# B&R Automation Studio project CrossCutterExercise
Automation Studio 4.12.4.107 SP; technology packages: Acp10Arnc0 5.24.1, mapp 5.24.1, mappView 5.24.1

## Configuration Config1

CPU 4PPC70.101G-20B, AutomationRuntime B4.93, Build 4.1.2, Safety 0.0, Vc V4.73.0

CPU 5PPC2100.BY22-000, AutomationRuntime B4.83, Build 4.1.2, Safety 0.0, Vc V4.73.0

CPU X20CP0484, AutomationRuntime B4.93, Build 4.1.2, Vc V4.72.6

### Task classes (Cpu.sw)
```
Cyclic#4:
  AxisCtrl <- SOURCE.Axis.AxisCtrl.prg
  VisuCtrl <- SOURCE.Visu.VisuCtrl.prg
  MainCtrl <- SOURCE.MainCtrl.prg
DataObjects: Acp10sys
NcDataObjects: acp10etxen <- acp10etxen.dob, gAxis01a <- gAxis01obj.gAxis01a.dob, gAxis01i <- gAxis01obj.gAxis01i.dob, gAxis02a <- gAxis02obj.gAxis02a.dob, gAxis02i <- gAxis02obj.gAxis02i.dob
Binaries: arsvcreg, udbdef, TCData, FWRules, Acp10map, acp10cfg, ashwd, ashwac, User, sysconf, asfw, arconfig, iomap, Role
Libraries: Acp10man, Acp10par, NcGlobal, Acp10_MC, sys_lib, brsystem, runtime, Acp10sim, MpAxis, MpBase, MpCom, powerlnk, astime, asbrstr, fileio, dataobj
```

### Hardware
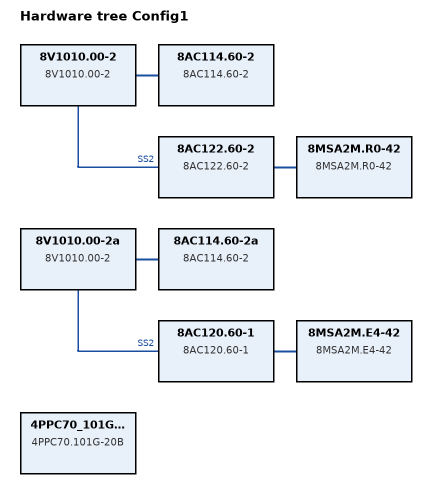
```
4PPC70_101G_20B : 4PPC70.101G-20B v1.5.4.0
  Connector IF2:
    ActivateDevice = 1
    Mode = Manual
    InternetAddress = 192.168.0.10
    SubnetMask = 255.255.255.0
    ActivateSnmp = 2
    DeviceParam = /EDDN=gei
  ConfigurationID = CrossCutterExercise_Config1
  PermanentPvSize = 2000
  RemanentGlobalPvSize = 2000
  TimerDeviceType = EPLX2X
  TimerDevice = 4PPC70_101G_20B.IF1
  TaskClassIdleTime = 2000
  FileDevice1
  FileDeviceName1 = USER
  FileDevicePath1 = USER_PATH
  KeyMappingFile = VC\4PPC70_101G_20B.dis
8AC114.60-2 : 8AC114.60-2 v1.0.0.8  [SS -> 8V1010.00-2.SS1; PLK1 -> 4PPC70_101G_20B.IF1 (NodeNumber=1) [Cable Type=PowerlinkCable, Length=10, Version=1.0.0.3]; PLK2 -> 8AC114.60-2a.PLK2 (NodeNumber=1) [Cable Type=PowerlinkCable, Length=10, Version=1.0.0.3]]
8AC114.60-2a : 8AC114.60-2 v1.0.0.8  [SS -> 8V1010.00-2a.SS1; PLK2 -> 8AC114.60-2.PLK2 (NodeNumber=2) [Cable Type=PowerlinkCable, Length=10, Version=1.0.0.3]]
8AC120.60-1 : 8AC120.60-1 v2.2.0.0  [SS -> 8V1010.00-2a.SS2]
8AC122.60-2 : 8AC122.60-2 v2.2.0.0  [SS -> 8V1010.00-2.SS2]
8MSA2M.E4-42 : 8MSA2M.E4-42 v1.0.0.0  [EC -> 8AC120.60-1.EC; MT -> 8V1010.00-2a.MT1]
8MSA2M.R0-42 : 8MSA2M.R0-42 v1.0.0.0  [EC -> 8AC122.60-2.EC; MT -> 8V1010.00-2.MT1]
8V1010.00-2 : 8V1010.00-2 v2.2.0.0
  MotionTP = Acp10Arnc0
  SinglePhaseOperation = on
  AxisIsPeriodic_r1 = on
  Period_r1 = 3600
  BothEndSwitchesAreNormallyOpen_r1 = on
  QuickStopIsNormallyOpen_r1 = on
8V1010.00-2a : 8V1010.00-2 v2.2.0.0
  MotionTP = Acp10Arnc0
  SinglePhaseOperation = on
  AxisIsPeriodic_r1 = on
  Period_r1 = 3600
  BothEndSwitchesAreNormallyOpen_r1 = on
  QuickStopIsNormallyOpen_r1 = on
```

### Acp10cfg.ncc - 4PPC70_101G_20B/Motion/Acp10cfg.ncc
```
NcConfiguration (Version=5.24.1, NcSwId=Acp10)
  ACP10CF1_typ:
    cnt_nettrc_rec_drive = 1500
    bufsize_trace_upload = 1200
    tc_nc_man_task = Cyclic #1
    glob_pv_as_ncobject = Yes
    ncsys_dl_broadcast = Yes
    ncsys_dl_acp_reset = Yes
    safemc_log_err_to_ax = Yes
    network_init:
      ncsw_init_execute = Yes
      automatic_execute = Yes
      node_nr_warning = Yes
      net_err_before_ncact = Yes
    nettrc:
      enter_parsecrec = Yes
      enter_ncaction = Yes
      save_ring_startidx = Yes
    cam_prof_download:
      cam_dat_dl_parallel = No
      tc_cam_dl_parallel = Task class for NC Manager task
    plk_if[0]:
      if_name = IF1
      tc_CycDat_PLCopen = Task class for NC Manager task
      mc_broadcast_extdat = No
```

### Acp10map.ncm - 4PPC70_101G_20B/Motion/Acp10map.ncm
```
NcMapping (NcSwId=Acp10, DisabledNodesAreHidden=False)
  NcObject gAxis02 (ModuleId=8V1010.00-2a, Type=ncAXIS, Channel=1, AcoposSimulation=Off, InitParameter=gAxis02i, AcoposParameter=gAxis02a, AdditionalData=PLCopen_ModPos="3600,1" , Disabled=FALSE, ModuleDisabled=FALSE)  // Master Axis
  NcObject gAxis01 (ModuleId=8V1010.00-2, Type=ncAXIS, Channel=1, AcoposSimulation=Off, InitParameter=gAxis01i, AcoposParameter=gAxis01a, AdditionalData=PLCopen_ModPos="3600,1" , Disabled=FALSE, ModuleDisabled=FALSE)  // Slave Axis
  NcObject 8V1010.00-2_ncV_AXIS1 (ModuleId=8V1010.00-2, Type=ncV_AXIS, Channel=1, Disabled=TRUE, ModuleDisabled=FALSE)
  NcObject 8V1010.00-2a_ncV_AXIS1 (ModuleId=8V1010.00-2a, Type=ncV_AXIS, Channel=1, Disabled=TRUE, ModuleDisabled=FALSE)
```

### Config.mpaxisbasic - 4PPC70_101G_20B/Motion/Config.mpaxisbasic
```
Element gML_Master (Type=mpaxisbasic)
```

### Config_1.mpaxisbasic - 4PPC70_101G_20B/Motion/Config_1.mpaxisbasic
```
Element gML_Slave (Type=mpaxisbasic)
  Alarms = MpAlarmX
```

### Config_4.mpaudittrail - 4PPC70_101G_20B/mappServices/Audit/Config_4.mpaudittrail
```
Element gAuditTrail (Type=mpaudittrail)
  Audit:
    Events:
      [0] = 16
      [1] = 2
      [2] = 18
    TextSource = TXT
      OutputFormat = Audit/Root
  Monitor:
    0:
      pv = ::VisuCtrl:SpeedInRPM
  Alarms = MpAlarmX
```

### Config_2.mpalarmxcore - 4PPC70_101G_20B/mappServices/Config_2.mpalarmxcore
```
Element gAlarmXCore (Type=mpalarmxcore)
  mapp.AlarmX.Core.Configuration:
    [0]:
      Name = EStopActive
      Message = Emergency Stop is Pressed
      Behavior = PersistentAlarm
```

### Config_4.mpaudittrail - 4PPC70_101G_20B/mappServices/Config_4.mpaudittrail
```
Element gAuditTrail (Type=mpaudittrail)
  Audit:
    Events:
      [0] = 16
      [1] = 2
      [2] = 18
```

### Config_5.mpcomgroup - 4PPC70_101G_20B/mappServices/Config_5.mpcomgroup
```
Element gGroup (Type=mpcomgroup)
  Linking:
    Subnodes:
      0 = gML_Master
      1 = gML_Slave
      2 = gAlarmXCore
  Alarms = MpAlarmX
Element gGroup_1 (Type=mpcomgroup)
  Linking:
    Subnodes:
      0 = gGroup
  Alarms = MpAlarmX
```

### Config_3.mpreportcore - 4PPC70_101G_20B/mappServices/Report/Config_3.mpreportcore
```
Element gReport (Type=mpreportcore)
  MpReport:
    PageLayouts:
      [0]:
        Name = Default
    Styles:
      Text:
        [0]:
          Name = Default
      Table:
        [0]:
          Name = Default
      Line:
        [0]:
          Name = Default
      Chart:
        PieChart:
          [0]:
            Name = Default
        LineChart:
          [0]:
            Name = Default
        BarChart:
          [0]:
            Name = Default
    Reports:
      [0]:
        PageLayout = Default
        [0]
```

### Config_6.mpuserx - 4PPC70_101G_20B/mappServices/User/Config_6.mpuserx
```
Element UserMgmtX (Type=mpuserx)
  ServerSettings:
    Server:
      AdditionalUserData:
        [0] = mail
        [1] = telephoneNumber
  Users:
    DefUser#1:
      id = Admin
      name = Admin
    DefUser#2:
      id = Anonymous
```

## Configuration CrossCutter

### Hardware
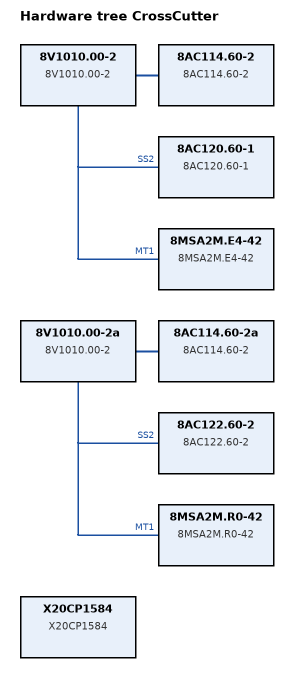
```
8AC114.60-2 : 8AC114.60-2 v1.0.0.8  [SS -> 8V1010.00-2.SS1; PLK1 -> X20CP1584.IF3 (NodeNumber=1) [Cable Type=PowerlinkCable, Length=10, Version=1.0.0.3]; PLK2 -> 8AC114.60-2a.PLK1 (NodeNumber=1) [Cable Type=PowerlinkCable, Length=10, Version=1.0.0.3]]
8AC114.60-2a : 8AC114.60-2 v1.0.0.8  [SS -> 8V1010.00-2a.SS1; PLK1 -> 8AC114.60-2.PLK2 (NodeNumber=2) [Cable Type=PowerlinkCable, Length=10, Version=1.0.0.3]]
8AC120.60-1 : 8AC120.60-1 v2.2.0.0  [SS -> 8V1010.00-2.SS2]
8AC122.60-2 : 8AC122.60-2 v2.2.0.0  [SS -> 8V1010.00-2a.SS2]
8MSA2M.E4-42 : 8MSA2M.E4-42 v1.0.0.0  [MT -> 8V1010.00-2.MT1]
8MSA2M.R0-42 : 8MSA2M.R0-42 v1.0.0.0  [MT -> 8V1010.00-2a.MT1]
8V1010.00-2 : 8V1010.00-2 v2.2.0.0
  MotionTP = Acp10Arnc0
  SinglePhaseOperation = on
  AxisIsPeriodic_r1 = on
  Period_r1 = 3600
  BothEndSwitchesAreNormallyOpen_r1 = on
  QuickStopIsNormallyOpen_r1 = on
8V1010.00-2a : 8V1010.00-2 v2.2.0.0
  MotionTP = Acp10Arnc0
  SinglePhaseOperation = on
  AxisIsPeriodic_r1 = on
  Period_r1 = 3600
  BothEndSwitchesAreNormallyOpen_r1 = on
  QuickStopIsNormallyOpen_r1 = on
X20CP1584 : X20CP1584 v1.10.0.0
  Connector IF2:
    ActivateDevice = 1
    Mode = Manual
    InternetAddress = 192.168.0.12
    SubnetMask = 255.255.255.0
    ActivateSnmp = 2
  ConfigurationID = CamAutomat_CrossCutter
  Simulation = 1
  TimerDeviceType = EPLX2X
  TimerDevice = X20CP1584.IF3
  TaskClassIdleTime = 2000
  FileDevice1
  FileDeviceName1 = USER
  FileDevicePath1 = USER_PATH
```

## Logical view

Binary libraries used (declarations not repeated): operator, runtime, astime, AsIecCon, sys_lib, brsystem, Acp10man, Acp10par, NcGlobal, Acp10sim 5.24.1, Acp10_MC, MpAxis 1.87.0, MpBase, MpCom 5.24.1, MpAlarmX, MpData, FileIO, DataObj, MpAudit 5.24.1, MpServer 5.24.0, MpUserX 5.24.1, MpReport 5.24.1

### Global.var - Global variables
```iecst
VAR
	gAxis01 : ACP10AXIS_typ; (*Slave Axis*)
	gAxis02 : ACP10AXIS_typ; (*Master Axis*)
	gVAxis01 : ACP10VAXIS_typ; (*Virtual Axis*)
	gVAxis02 : ACP10VAXIS_typ; (*Virtual Axis*)
	MpAxisSlave : MpAxisBasic; (*FB for Slave*)
	MpAxisMaster : MpAxisBasic; (*FB for Master*)
	MpAxisCamSequencer_0 : MpAxisCamSequencer; (*Cam Sequencer FB*)
	CamSeqPara : MpAxisCamSequencerParType; (*Cam Sequence Parameter*)
	SlavePara : MpAxisBasicParType; (*Slave Axis Parameter*)
	MasterPara : MpAxisBasicParType; (*Master Axis Parameter*)
END_VAR
```


### Data object Logical/acp10etxen (Ett)

- acp10etxen.ett (not shown)

### Package Logical/gAxis01obj - gAxis03obj

### gAxis01i.ax
```
InitParameter (Version=5.24.1, NcSwId=Acp10)
  ACP10AXIS_typ:
    dig_in:
      level:
        reference = ncACTIV_HI + ncFORCE
        pos_hw_end = ncACTIV_HI + ncFORCE
        neg_hw_end = ncACTIV_HI + ncFORCE
        trigger1 = ncACTIV_HI
        trigger2 = ncACTIV_HI
    encoder_if:
      parameter:
        count_dir = ncINVERSE
        scaling:
          load:
            units = 3600
            rev_motor = 1
    limit:
      parameter:
        v_pos = 50000.0
        v_neg = 50000.0
        a1_pos = 120000.0
        a2_pos = 120000.0
        a1_neg = 120000.0
        a2_neg = 120000.0
        t_jolt = 0.02
        t_in_pos = 0
        pos_sw_end = 2000000000
        neg_sw_end = -2000000000
        ds_warning = 500
        ds_stop = 1000
        a_stop = 1.0e30
        dv_stop = 0
        dv_stop_mode = ncOFF
    controller:
      mode = ncPOSITION
      position:
        kv = 50
        tn = 0
        t_predict = 0.0004
        t_total = 0.0004
        p_max = 1.0e30
        i_max = 0
      speed:
        kv = 0.2
        tn = 0
        t_filter = 0.0
        isq_filter1:
          type = ncOFF
          a0 = 0.0
          a1 = 0.0
          b0 = 0.0
          b1 = 0.0
          b2 = 0.0
          c0_par_id = 0
          c1_par_id = 0
        isq_filter2:
          type = ncOFF
          a0 = 0.0
          a1 = 0.0
          b0 = 0.0
          b1 = 0.0
          b2 = 0.0
          c0_par_id = 0
          c1_par_id = 0
        isq_filter3:
          type = ncOFF
          a0 = 0.0
          a1 = 0.0
          b0 = 0.0
          b1 = 0.0
          b2 = 0.0
          c0_par_id = 0
          c1_par_id = 0
      uf:
        type = ncLINEAR + ncCORRECTION
        auto_config = ncMOTOR_PAR
        u0 = 0
        un = 0
        fn = 50.0
        k_f_slip = 0
      ff:
        mode = ncSTANDARD
        torque_load = 0.0
        torque_pos = 0.0
        torque_neg = 0.0
        kv_torque = 0.0
        inertia = 0.0
        t_filter_a = 0.0
      fb:
        mode = ncSTANDARD
        speed_mix_ratio = 0.0
        speed_kv = 0.2
      model:
        mass1:
          inertia = 0
          viscous_friction = 0
        mass2:
          inertia = 0
          viscous_friction = 0
          stiffness = 0
          damping = 0
    move:
      stop:
        parameter[0]:
          decel_ramp = ncA_LIMIT
          controller = ncON
        parameter[1]:
          decel_ramp = ncA_LIMIT
          controller = ncON
        parameter[2]:
          decel_ramp = ncA_LIMIT
          controller = ncON
        parameter[3]:
          decel_ramp = ncA_LIMIT
          controller = ncON
        quickstop:
          decel_ramp = ncA_LIMIT
          t_jolt = 0
        drive_error:
          decel_ramp = ncA_LIMIT
      homing:
        parameter:
          s = 0
          v_switch = 5000
          v_trigger = 500
          a = 50000
          mode = ncDIRECT
          edge_sw = ncPOSITIVE
          start_dir = ncPOSITIVE
          trigg_dir = ncPOSITIVE
          ref_pulse = ncOFF
          fix_dir = ncOFF
          tr_s_block = 0
          torque_lim = 0
          ds_block = 0
          ds_stop = 0
      basis:
        parameter:
          v_pos = 5000
          v_neg = 5000
          a1_pos = 50000
          a2_pos = 50000
          a1_neg = 50000
          a2_neg = 50000
    message:
      text:
        parameter:
          format = ncBREAK
          columns = 80
          data_modul = acp10etxen
```

### Package Logical/gAxis02obj - gAxis04obj

### gAxis02i.ax
```
InitParameter (Version=5.24.1, NcSwId=Acp10)
  ACP10AXIS_typ:
    dig_in:
      level:
        reference = ncACTIV_HI + ncFORCE
        pos_hw_end = ncACTIV_HI + ncFORCE
        neg_hw_end = ncACTIV_HI + ncFORCE
        trigger1 = ncACTIV_HI
        trigger2 = ncACTIV_HI
    encoder_if:
      parameter:
        count_dir = ncINVERSE
        scaling:
          load:
            units = 3600
            rev_motor = 1
    limit:
      parameter:
        v_pos = 50000.0
        v_neg = 50000.0
        a1_pos = 120000.0
        a2_pos = 120000.0
        a1_neg = 120000.0
        a2_neg = 120000.0
        t_jolt = 0.02
        t_in_pos = 0
        pos_sw_end = 2000000000
        neg_sw_end = -2000000000
        ds_warning = 500
        ds_stop = 1000
        a_stop = 1.0e30
        dv_stop = 0
        dv_stop_mode = ncOFF
    controller:
      mode = ncPOSITION
      position:
        kv = 50
        tn = 0
        t_predict = 0.0044
        t_total = 0.0044
        p_max = 1.0e30
        i_max = 0
      speed:
        kv = 0.2
        tn = 0
        t_filter = 0.0
        isq_filter1:
          type = ncOFF
          a0 = 0.0
          a1 = 0.0
          b0 = 0.0
          b1 = 0.0
          b2 = 0.0
          c0_par_id = 0
          c1_par_id = 0
        isq_filter2:
          type = ncOFF
          a0 = 0.0
          a1 = 0.0
          b0 = 0.0
          b1 = 0.0
          b2 = 0.0
          c0_par_id = 0
          c1_par_id = 0
        isq_filter3:
          type = ncOFF
          a0 = 0.0
          a1 = 0.0
          b0 = 0.0
          b1 = 0.0
          b2 = 0.0
          c0_par_id = 0
          c1_par_id = 0
      uf:
        type = ncLINEAR + ncCORRECTION
        auto_config = ncMOTOR_PAR
        u0 = 0
        un = 0
        fn = 50.0
        k_f_slip = 0
      ff:
        mode = ncSTANDARD
        torque_load = 0.0
        torque_pos = 0.0
        torque_neg = 0.0
        kv_torque = 0.0
        inertia = 0.0
        t_filter_a = 0.0
      fb:
        mode = ncSTANDARD
        speed_mix_ratio = 0.0
        speed_kv = 2.0
      model:
        mass1:
          inertia = 0
          viscous_friction = 0
        mass2:
          inertia = 0
          viscous_friction = 0
          stiffness = 0
          damping = 0
    move:
      stop:
        parameter[0]:
          decel_ramp = ncA_LIMIT
          controller = ncON
        parameter[1]:
          decel_ramp = ncA_LIMIT
          controller = ncON
        parameter[2]:
          decel_ramp = ncA_LIMIT
          controller = ncON
        parameter[3]:
          decel_ramp = ncA_LIMIT
          controller = ncON
        quickstop:
          decel_ramp = ncA_LIMIT
          t_jolt = 0
        drive_error:
          decel_ramp = ncA_LIMIT
      homing:
        parameter:
          s = 0
          v_switch = 5000
          v_trigger = 500
          a = 50000
          mode = ncDIRECT
          edge_sw = ncPOSITIVE
          start_dir = ncPOSITIVE
          trigg_dir = ncPOSITIVE
          ref_pulse = ncOFF
          fix_dir = ncOFF
          tr_s_block = 0
          torque_lim = 0
          ds_block = 0
          ds_stop = 0
      basis:
        parameter:
          v_pos = 5000
          v_neg = 5000
          a1_pos = 50000
          a2_pos = 50000
          a1_neg = 50000
          a2_neg = 50000
    message:
      text:
        parameter:
          format = ncBREAK
          columns = 80
          data_modul = acp10etxen
```

### Main.typ
```iecst
TYPE
	Main_typ : 	STRUCT
		Cmd : MainCmd_typ;
		Status : MainStatus_typ;
	END_STRUCT;
	MainCmd_typ : 	STRUCT
		bStart : BOOL;
		bStop : BOOL;
		bEStop : BOOL;
	END_STRUCT;
	MainStatus_typ : 	STRUCT
	END_STRUCT;
END_TYPE
```

### Program Logical/SOURCE/MainCtrl (IEC)

#### Types.typ
```iecst
TYPE
	eMainState :
		(
		WAIT,
		SELECT_MODE,
		SINGLE_BLADE,
		DUAL_BLADE,
		ERROR
		);
END_TYPE
```

#### Variables.var
```iecst
VAR
	MainState : eMainState;
END_VAR
```

#### Main.st
```iecst
(*|ŻŻŻŻŻŻŻŻŻŻŻŻŻŻŻŻŻŻŻŻŻŻŻŻŻŻŻŻŻŻŻŻŻŻŻŻŻŻŻŻŻŻŻŻŻŻŻŻŻŻŻŻŻŻŻŻŻŻŻŻŻŻŻŻŻŻŻŻŻŻŻŻŻŻŻŻŻŻŻŻŻŻŻŻŻŻŻŻŻŻŻŻŻŻŻŻŻŻŻŻŻŻŻŻŻŻŻŻŻŻ|*)
(*| Copyright      :-  B&R Industrial Automation GmbH                                                            |*)
(*| Contact Person :-   salis                                                                          		     |*)
(*|——————————————————————————————————————————————————————————————————————————————————————————————————————————————|*)
(*| System       :-  Cross Cutter                                                                                |*)
(*| Task Name    :-  MainCtrl.st                                                                                 |*)
(*| Auther Name  :-   salis                                                                                      |*)
(*| Created Date :-  April 28, 2024/10:21 AM                                                                     |*)
(*| AS Version   :-  AS 4.12.4.107 SP                                                                            |*)
(*|——————————————————————————————————————————————————————————————————————————————————————————————————————————————|*)
(*| Description  :-  Main Control and Mode Selection Logic                                                       |*)
(*|                                                                                                              |*)
(*|——————————————————————————————————————————————————————————————————————————————————————————————————————————————|*)
(*| Version :-         V 1.0                      salis                                                          |*)
(*|——————————————————————————————————————————————————————————————————————————————————————————————————————————————|*)
PROGRAM _INIT

END_PROGRAM

PROGRAM _CYCLIC
	(********************************* State Machine for Main Control and Mode Selection ***************************************)

	CASE MainState OF
		WAIT:

			IF Main.Cmd.bStart THEN
				MainState := SELECT_MODE;
			END_IF

		SELECT_MODE:
			IF Main.Cmd.bSingleBlade THEN
				MainState := SINGLE_BLADE;
			ELSIF Main.Cmd.bDoubleBlade THEN
				MainState := DUAL_BLADE;
			END_IF
			MpAxisMaster.Update := FALSE;
			MpAxisSlave.Update := FALSE;

		SINGLE_BLADE:
			Main.Cmd.bDoubleBlade := FALSE;
			Axis.Cmd.bDoubleBlade := FALSE;
			Main.Cmd.bSingleBlade := FALSE;
			Axis.Cmd.bSingleBlade := TRUE;
			MpAxisMaster.Update := TRUE;
			MpAxisSlave.Update := TRUE;
			IF MpAxisMaster.UpdateDone AND MpAxisSlave.UpdateDone THEN
				MainState := SELECT_MODE;
			END_IF

		DUAL_BLADE:
			Main.Cmd.bSingleBlade := FALSE;
			Axis.Cmd.bSingleBlade := FALSE;
			Main.Cmd.bDoubleBlade := FALSE;
			Axis.Cmd.bDoubleBlade := TRUE;
			MpAxisMaster.Update := TRUE;
			MpAxisSlave.Update := TRUE;
			IF MpAxisMaster.UpdateDone AND MpAxisSlave.UpdateDone THEN
				MainState := SELECT_MODE;
			END_IF
	END_CASE;

END_PROGRAM

PROGRAM _EXIT

END_PROGRAM
```

### Axis.typ
```iecst
TYPE
	Axis_typ : 	STRUCT
		Cmd : AxisCmd_typ;
		Para : AxisPara_typ;
	END_STRUCT;
	AxisCmd_typ : 	STRUCT
		bStart : BOOL;
		bHome : BOOL;
		bStop : BOOL;
		bEStop : BOOL;
	END_STRUCT;
	AxisPara_typ : 	STRUCT
		gMachineSpeed : USINT;
	END_STRUCT;
END_TYPE
```

### Program Logical/SOURCE/Axis/AxisCtrl (IEC)

#### Main.st - Init, cyclic, exit code
```iecst
PROGRAM _INIT
	(* Insert code here *)
	MasterPara.Acceleration := 5000;
	MasterPara.Deceleration := 10000;

	MasterPara.Position := 0;

	SlavePara.Acceleration := 5000;
	SlavePara.Deceleration := 10000;

	SlavePara.Position := 0;;

END_PROGRAM

PROGRAM _CYCLIC
	(* Insert code here *)

	MpAxisMaster.MpLink := ADR(gML_Master);
	MpAxisMaster.Enable := TRUE;
	MpAxisMaster.Parameters := ADR(MasterPara);
	MpAxisMaster.Axis := ADR(gAxis02);
	MpAxisMaster();

	MpAxisSlave.MpLink := ADR(gML_Slave);
	MpAxisSlave.Enable := TRUE;
	MpAxisSlave.Parameters := ADR(SlavePara);
	MpAxisSlave.Axis := ADR(gAxis01);
	MpAxisSlave();

	SingleBladeCam;

	MpAxisCamSequencer_0.MpLink := ADR(gML_Slave);
	MpAxisCamSequencer_0.MpLinkMaster := ADR(gML_Master);
	MpAxisCamSequencer_0.Enable := TRUE;
	MpAxisCamSequencer_0.Parameters := ADR(CamSeqPara);
	MpAxisCamSequencer_0();

	IF Axis.Cmd.bHome THEN
		MasterPara.Direction := mpAXIS_DIR_SHORTEST_WAY;
		SlavePara.Direction := mpAXIS_DIR_SHORTEST_WAY;
		MasterPara.Velocity := 1200;
		SlavePara.Velocity := 1200;
	ELSE
		MasterPara.Direction := mpAXIS_DIR_POSITIVE;
		SlavePara.Direction := mpAXIS_DIR_POSITIVE;
		MasterPara.Velocity := 3600;
		SlavePara.Velocity := 3600;
	END_IF

//	IF (MpAxisMaster.Position <= 1560) AND (MpAxisMaster.Position >= 2060) THEN
//		MpAxisMaster.Power := FALSE;
//		MpAxisSlave.Power := FALSE;
//	ELSIF MpAxisMaster.Active AND MpAxisSlave.Active THEN
//		MpAxisMaster.Power := TRUE;
//		MpAxisSlave.Power := TRUE;
//	END_IF

	CASE AxisHomeState OF
		WAIT:
			IF (MpAxisMaster.Power = TRUE) AND (MpAxisSlave.Power = TRUE) THEN
				IF Axis.Cmd.bHome THEN
					AxisHomeState := HOME;
				END_IF
			END_IF
		HOME:
			MpAxisCamSequencer_0.StartSequence := FALSE;
			MpAxisMaster.MoveAbsolute := TRUE;
			MpAxisSlave.MoveAbsolute := TRUE;
			IF (MpAxisMaster.Position = MasterPara.Position) AND (MpAxisSlave.Position = SlavePara.Position) THEN
				AxisHomeState := HOMING_ACTIVE;
			END_IF

		HOMING_ACTIVE:
			MpAxisMaster.MoveAbsolute := FALSE;
			MpAxisSlave.MoveAbsolute := FALSE;
			MpAxisMaster.Home := TRUE;
			MpAxisSlave.Home := TRUE;
			IF MpAxisMaster.IsHomed AND MpAxisSlave.IsHomed THEN
				AxisHomeState := HOME_OK;
			END_IF

		HOME_OK:
			MpAxisCamSequencer_0.StartSequence := TRUE;
			Axis.Cmd.bHome := FALSE;
			MpAxisMaster.MoveAbsolute := FALSE;
			MpAxisSlave.MoveAbsolute := FALSE;
			MpAxisMaster.Home := FALSE;
			MpAxisSlave.Home := FALSE;
			AxisHomeState := WAIT;

	END_CASE;

END_PROGRAM

PROGRAM _EXIT
	(* Insert code here *)

END_PROGRAM
```

#### Types.typ - Local data types
```iecst
TYPE
	eAxisHome :
		(
		WAIT,
		HOMING_ACTIVE,
		HOME,
		HOME_OK,
		ERROR
		);
END_TYPE
```

#### Variables.var - Local variables
```iecst
VAR
	AxisHomeState : eAxisHome;
	Axis : Axis_typ;
END_VAR
```

#### SingleBladeCam.st - Cam logic for single blade cross cutter
```iecst
ACTION SingleBladeCam:
	CamSeqPara.Configuration.Master 			:= ADR(gAxis02);
	CamSeqPara.Configuration.MasterParID 		:= ACP10PAR_PCTRL_S_ACT;

	(** Event 0 - WAIT FOR TRIGGER **)
	CamSeqPara.Configuration.State[0].Event[0].Type 				:= ncST_END; //Trigger
	CamSeqPara.Configuration.State[0].Event[0].Attribute		 	:= ncST_END; //Reaction
	CamSeqPara.Configuration.State[0].Event[0].NextState 			:= 1; //Next State
	(*************************** STATE 1 ****************************)
	CamSeqPara.Configuration.State[1].CamProfileIndex 		  		:= 16#FFFE;
	CamSeqPara.Configuration.State[1].MasterFactor 					:= 1; //Master Dist.
	CamSeqPara.Configuration.State[1].SlaveFactor 					:= 1; //Slave Dist.

	CamSeqPara.Configuration.State[1].CompMode   	 				:= ncONLYCOMP;
	CamSeqPara.Configuration.State[1].MasterCompDistance			:= 1620; //Master Dist.
	CamSeqPara.Configuration.State[1].SlaveCompDistance				:= 1620; //Slave Dist.

	(** Event **)
	CamSeqPara.Configuration.State[1].Event[0].Type 				:= ncST_END; //Trigger
	CamSeqPara.Configuration.State[1].Event[0].Attribute 			:= ncST_END; //Reaction
	CamSeqPara.Configuration.State[1].Event[0].NextState 			:= 2; //Next State

	(*************************** STATE 2 ****************************)
	CamSeqPara.Configuration.State[2].CamProfileIndex 				:= 16#FFFF;
	CamSeqPara.Configuration.State[2].MasterFactor 					:= 360;  //Master Dist.
	CamSeqPara.Configuration.State[2].SlaveFactor 					:= -360; //Slave Dist.

	(** Event **)
	CamSeqPara.Configuration.State[2].Event[0].Type 				:= ncST_END; //Trigger
	CamSeqPara.Configuration.State[2].Event[0].Attribute 			:= ncST_END; //Reaction
	CamSeqPara.Configuration.State[2].Event[0].NextState 			:= 3; //Next State

	(*************************** STATE 3 ****************************)
	CamSeqPara.Configuration.State[3].CamProfileIndex 				:= 16#FFFE;
	CamSeqPara.Configuration.State[3].MasterFactor 					:= 1; //Master Dist.
	CamSeqPara.Configuration.State[3].SlaveFactor 					:= 1; //Slave Dist.

	CamSeqPara.Configuration.State[3].CompMode   	 				:= ncONLYCOMP;
	CamSeqPara.Configuration.State[3].MasterCompDistance			:= 1620; //Master Dist.
	CamSeqPara.Configuration.State[3].SlaveCompDistance				:= 1620; //Slave Dist.

	(** Event **)
	CamSeqPara.Configuration.State[3].Event[0].Type 				:= ncST_END; //Trigger
	CamSeqPara.Configuration.State[3].Event[0].Attribute 			:= ncST_END; //Reaction
	CamSeqPara.Configuration.State[3].Event[0].NextState 			:= 1; //Next State
END_ACTION
```

#### DoubleBladeCam.st - Cam logic for Double blade cross cutter
```iecst
ACTION DoubleBladeCam:

	CamSeqPara.Configuration.Master 			:= ADR(gAxis02);
	CamSeqPara.Configuration.MasterParID 		:= ACP10PAR_PCTRL_S_ACT;

	(** Event 0 - WAIT FOR TRIGGER **)
	CamSeqPara.Configuration.State[0].Event[0].Type 				:= ncST_END; //Trigger
	CamSeqPara.Configuration.State[0].Event[0].Attribute		 	:= ncST_END; //Reaction
	CamSeqPara.Configuration.State[0].Event[0].NextState 			:= 1; //Next State
	(*************************** STATE 1 ****************************)
	CamSeqPara.Configuration.State[1].CamProfileIndex 		  		:= 16#FFFE;
	CamSeqPara.Configuration.State[1].MasterFactor 					:= 1; //Master Dist.
	CamSeqPara.Configuration.State[1].SlaveFactor 					:= 1; //Slave Dist.

	CamSeqPara.Configuration.State[1].CompMode   	 				:= ncONLYCOMP;
	CamSeqPara.Configuration.State[1].MasterCompDistance			:= 1580; //Master Dist.
	CamSeqPara.Configuration.State[1].SlaveCompDistance				:= 1580; //Slave Dist.

	(** Event **)
	CamSeqPara.Configuration.State[1].Event[0].Type 				:= ncST_END; //Trigger
	CamSeqPara.Configuration.State[1].Event[0].Attribute 			:= ncST_END; //Reaction
	CamSeqPara.Configuration.State[1].Event[0].NextState 			:= 2; //Next State

	(*************************** STATE 2 ****************************)
	CamSeqPara.Configuration.State[2].CamProfileIndex 				:= 16#FFFF;
	CamSeqPara.Configuration.State[2].MasterFactor 					:= 400;  //Master Dist.
	CamSeqPara.Configuration.State[2].SlaveFactor 					:= -400; //Slave Dist.

	(** Event **)
	CamSeqPara.Configuration.State[2].Event[0].Type 				:= ncST_END; //Trigger
	CamSeqPara.Configuration.State[2].Event[0].Attribute 			:= ncST_END; //Reaction
	CamSeqPara.Configuration.State[2].Event[0].NextState 			:= 0; //Next State

	(*************************** STATE 3 ****************************)
	CamSeqPara.Configuration.State[3].CamProfileIndex 				:= 16#FFFE;
	CamSeqPara.Configuration.State[3].MasterFactor 					:= 1; //Master Dist.
	CamSeqPara.Configuration.State[3].SlaveFactor 					:= 1; //Slave Dist.

	CamSeqPara.Configuration.State[3].CompMode   	 				:= ncONLYCOMP;
	CamSeqPara.Configuration.State[3].MasterCompDistance			:= 1620; //Master Dist.
	CamSeqPara.Configuration.State[3].SlaveCompDistance				:= 1620; //Slave Dist.

	(** Event **)
	CamSeqPara.Configuration.State[3].Event[0].Type 				:= ncST_END; //Trigger
	CamSeqPara.Configuration.State[3].Event[0].Attribute 			:= ncST_END; //Reaction
	CamSeqPara.Configuration.State[3].Event[0].NextState 			:= 4; //Next State

	(*************************** STATE 4 ****************************)
	CamSeqPara.Configuration.State[4].CamProfileIndex 				:= 16#FFFF;
	CamSeqPara.Configuration.State[4].MasterFactor 					:= 360;  //Master Dist.
	CamSeqPara.Configuration.State[4].SlaveFactor 					:= -360; //Slave Dist.

	(** Event **)
	CamSeqPara.Configuration.State[4].Event[0].Type 				:= ncST_END; //Trigger
	CamSeqPara.Configuration.State[4].Event[0].Attribute 			:= ncST_END; //Reaction
	CamSeqPara.Configuration.State[4].Event[0].NextState 			:= 1; //Next State
END_ACTION
```

### Axis.var - not listed in the package file held
```iecst
VAR
	Axis : Axis_typ;
END_VAR
VAR CONSTANT
	SPositionSingle : INT := 3550;
	MPositionSingle : INT := 3450;
	SlaveOffsetSingle : INT := 0;
	MasterOffsetSingle : INT := 0;
	MUpPositionDouble : INT := 825;
	SPositionDouble : INT := 2225;
	MDownPositionDouble : INT := 2625;
	MasterUpOffsetDouble : INT := 825;
	MasterDownOffsetDouble : INT := 2625;
	HomingVelocity : INT := 1200;
	MUpPosLimit1 : INT := 1480;
	MUpPosLimit2 : INT := 3501;
	MUpNegLimit1 : INT := 0;
	MUpNegLimit2 : INT := 3599;
	MDownNegLimit : INT := 1940;
	MDownPosLimit : INT := 3500;
	MCutRegionNegLimit1 : INT := 1480;
	MCutRegionPosLimit1 : INT := 1940;
	MCutRegionNegLimit2 : INT := 3280;
	MCutRegionPosLimit2 : INT := 3599;
	MCutRegionPosLimit3 : INT := 1;
	MCutRegionNegLimit3 : INT := 150;
	RunDeceleration : UDINT := 72000;
	RunAcceleration : UDINT := 72000;
	HomeAcceleration : UDINT := 3600;
	HomeVelocity : UDINT := 720;
	JogVelocity : UDINT := 7200;
END_VAR
```

- Visualisation Logical/SOURCE/Visu (not shown)

### Main.var - not listed in the package file held
```iecst
VAR
	Main : Main_typ;
	MachineStatus : STRING[80];
END_VAR
```

### Program Logical/SOURCE/Alarm/AlarmCtrl (IEC) - Program for Alarm

#### Variables.var
```iecst
VAR
	MpAlarm : MpAlarmXCore;
END_VAR
```

#### Main.st
```iecst
(*|ŻŻŻŻŻŻŻŻŻŻŻŻŻŻŻŻŻŻŻŻŻŻŻŻŻŻŻŻŻŻŻŻŻŻŻŻŻŻŻŻŻŻŻŻŻŻŻŻŻŻŻŻŻŻŻŻŻŻŻŻŻŻŻŻŻŻŻŻŻŻŻŻŻŻŻŻŻŻŻŻŻŻŻŻŻŻŻŻŻŻŻŻŻŻŻŻŻŻŻŻŻŻŻŻŻŻŻŻŻŻ|*)
(*| Copyright      :-  B&R Industrial Automation GmbH                                                            |*)
(*| Contact Person :-   salis                                                                          		     |*)
(*|——————————————————————————————————————————————————————————————————————————————————————————————————————————————|*)
(*| System       :-  Cross Cutter                                                                                |*)
(*| Task Name    :-  AlarmCtrl.st                                                                                |*)
(*| Auther Name  :-   salis                                                                                      |*)
(*| Created Date :-  April 28, 2024/10:21 AM                                                                     |*)
(*| AS Version   :-  AS 4.12.4.107 SP                                                                            |*)
(*|——————————————————————————————————————————————————————————————————————————————————————————————————————————————|*)
(*| Description  :-  Alarm Control Logic                               											 |*)
(*|                                                                                                              |*)
(*|——————————————————————————————————————————————————————————————————————————————————————————————————————————————|*)
(*| Version :-         V 1.0                      salis                                                          |*)
(*|——————————————————————————————————————————————————————————————————————————————————————————————————————————————|*)
PROGRAM _INIT
	(* Insert code here *)

END_PROGRAM

PROGRAM _CYCLIC
	(********************************* Function block for Alarm ***************************************)

	MpAlarm(MpLink := ADR(gAlarmXCore) , Enable := TRUE);
END_PROGRAM

PROGRAM _EXIT
	(* Insert code here *)

END_PROGRAM
```

### Program Logical/SOURCE/Audit/Audit (IEC)

#### Variables.var
```iecst
VAR
	MpAuditRegPar_0 : MpAuditRegPar;
	MpAuditTrail_0 : MpAuditTrail;
END_VAR
```

#### Main.st
```iecst
(*|ŻŻŻŻŻŻŻŻŻŻŻŻŻŻŻŻŻŻŻŻŻŻŻŻŻŻŻŻŻŻŻŻŻŻŻŻŻŻŻŻŻŻŻŻŻŻŻŻŻŻŻŻŻŻŻŻŻŻŻŻŻŻŻŻŻŻŻŻŻŻŻŻŻŻŻŻŻŻŻŻŻŻŻŻŻŻŻŻŻŻŻŻŻŻŻŻŻŻŻŻŻŻŻŻŻŻŻŻŻŻ|*)
(*| Copyright      :-  B&R Industrial Automation GmbH                                                            |*)
(*| Contact Person :-   salis                                                                          		     |*)
(*|——————————————————————————————————————————————————————————————————————————————————————————————————————————————|*)
(*| System       :-  Cross Cutter                                                                                |*)
(*| Task Name    :-  Audit.st                                                                                    |*)
(*| Auther Name  :-   salis                                                                                      |*)
(*| Created Date :-  April 28, 2024/10:21 AM                                                                     |*)
(*| AS Version   :-  AS 4.12.4.107 SP                                                                            |*)
(*|——————————————————————————————————————————————————————————————————————————————————————————————————————————————|*)
(*| Description  :-  Audit Control Logic                               											 |*)
(*|                                                                                                              |*)
(*|——————————————————————————————————————————————————————————————————————————————————————————————————————————————|*)
(*| Version :-         V 1.0                      salis                                                          |*)
(*|——————————————————————————————————————————————————————————————————————————————————————————————————————————————|*)
PROGRAM _INIT
	(* Insert code here *)

END_PROGRAM

PROGRAM _CYCLIC
	(********************************* Function Block For Audit and Event Log ***************************************)

	MpAuditRegPar_0(MpLink := ADR(gAuditTrail), Enable := TRUE, PVName := ADR('VisuCtrl:SpeedInRPM') );

	MpAuditTrail_0(MpLink := ADR(gAuditTrail), Enable := TRUE, Language := ADR('en'), DeviceName := ADR('Audit'));
END_PROGRAM

PROGRAM _EXIT
	(* Insert code here *)

END_PROGRAM
```

### Program Logical/AxisCtrl (IEC)

#### Main.st - Init, cyclic, exit code
```iecst
PROGRAM _INIT
	(* Insert code here *)
	MasterPara.Acceleration := 5000;
	MasterPara.Deceleration := 10000;
	MasterPara.Velocity := 3600;
	SlavePara.Acceleration := 5000;
	SlavePara.Deceleration := 10000;
	SlavePara.Velocity := 3600;

END_PROGRAM

PROGRAM _CYCLIC
	(* Insert code here *)

	MpAxisMaster.MpLink := ADR(gML_Master);
	MpAxisMaster.Enable := TRUE;
	MpAxisMaster.Parameters := ADR(MasterPara);
	MpAxisMaster.Axis := ADR(gAxis04);
	MpAxisMaster();

	MpAxisSlave.MpLink := ADR(gML_Slave);
	MpAxisSlave.Enable := TRUE;
	MpAxisSlave.Parameters := ADR(SlavePara);
	MpAxisSlave.Axis := ADR(gAxis03);
	MpAxisSlave();

	Exercise4;

	MpAxisCamSequencer_0.MpLink := ADR(gML_Slave);
	MpAxisCamSequencer_0.MpLinkMaster := ADR(gML_Master);
	MpAxisCamSequencer_0.Enable := TRUE;
	MpAxisCamSequencer_0.Parameters := ADR(CamSeqPara);
	MpAxisCamSequencer_0();

//	MasterPosition := LREAL_TO_UDINT(MpAxisMaster.Position) MOD 3600;
//	IF (MasterPosition >= 600) AND (MasterPosition < 900) THEN
//		gMi_Signal1 := TRUE;
//	ELSIF (MasterPosition >= 900) THEN
//		gMi_Signal1 := FALSE;
//	END_IF
//

//	CASE MasterState OF
//		PowerOn:
//			IF MpAxisMaster.Active THEN
//				MpAxisMaster.Power := TRUE;
//			END_IF
//			IF MpAxisMaster.PowerOn THEN
//				MasterState := Home;
//			END_IF
//		Home:
//			MpAxisMaster.Home := TRUE;
//			IF MpAxisMaster.IsHomed THEN
//				MasterState := HomingOk;
//			END_IF
//		HomingOk:
//			MpAxisMaster.Home := FALSE;
//	END_CASE
//
//	CASE SlaveState OF
//		PowerOn:
//			IF MpAxisSlave.Active THEN
//				MpAxisSlave.Power := TRUE;
//			END_IF
//			IF MpAxisSlave.PowerOn THEN
//				SlaveState := Home;
//			END_IF
//		Home:
//			MpAxisSlave.Home := TRUE;
//			IF MpAxisSlave.IsHomed THEN
//				SlaveState := HomingOk;
//			END_IF
//		HomingOk:
//			MpAxisSlave.Home := FALSE;
//	END_CASE
//
//	IF MpAxisMaster.IsHomed AND MpAxisSlave.IsHomed THEN
//		MpAxisCamSequencer_0.StartSequence := TRUE;
//	END_IF
END_PROGRAM

PROGRAM _EXIT
	(* Insert code here *)

END_PROGRAM
```

#### Types.typ - Local data types
```iecst
TYPE
	eAxis :
		(
		PowerOn,
		Home,
		HomingOk
		);
END_TYPE
```

#### Variables.var - Local variables
```iecst
VAR
	MpAxisSlave : MpAxisBasic;
	MpAxisMaster : MpAxisBasic;
	MpAxisCamSequencer_0 : MpAxisCamSequencer;
	CamSeqPara : MpAxisCamSequencerParType;
	SlavePara : MpAxisBasicParType;
	MasterPara : MpAxisBasicParType;
	SlaveState : eAxis;
	MasterState : eAxis;
END_VAR
```

#### Exercise4.st
```iecst
ACTION Exercise4:
	CamSeqPara.Configuration.Master 			:= ADR(gAxis04);
	CamSeqPara.Configuration.MasterParID 		:= ACP10PAR_PCTRL_S_ACT;

	(** Event 0 - WAIT FOR TRIGGER **)
	CamSeqPara.Configuration.State[0].Event[0].Type 				:= ncST_END; //Trigger
	CamSeqPara.Configuration.State[0].Event[0].Attribute		 	:= ncST_END; //Reaction
	CamSeqPara.Configuration.State[0].Event[0].NextState 			:= 1; //Next State
	(*************************** STATE 1 ****************************)
	CamSeqPara.Configuration.State[1].CamProfileIndex 		  		:= 16#FFFE;
	CamSeqPara.Configuration.State[1].MasterFactor 					:= 1; //Master Dist.
	CamSeqPara.Configuration.State[1].SlaveFactor 					:= 1; //Slave Dist.

	CamSeqPara.Configuration.State[1].CompMode   	 				:= ncONLYCOMP;
	CamSeqPara.Configuration.State[1].MasterCompDistance			:= 1620; //Master Dist.
	CamSeqPara.Configuration.State[1].SlaveCompDistance				:= 1620; //Slave Dist.

	(** Event **)
	CamSeqPara.Configuration.State[1].Event[0].Type 				:= ncST_END; //Trigger
	CamSeqPara.Configuration.State[1].Event[0].Attribute 			:= ncST_END; //Reaction
	CamSeqPara.Configuration.State[1].Event[0].NextState 			:= 2; //Next State

	(*************************** STATE 2 ****************************)
	CamSeqPara.Configuration.State[2].CamProfileIndex 				:= 16#FFFF;
	CamSeqPara.Configuration.State[2].MasterFactor 					:= 360;  //Master Dist.
	CamSeqPara.Configuration.State[2].SlaveFactor 					:= -360; //Slave Dist.

	(** Event **)
	CamSeqPara.Configuration.State[2].Event[0].Type 				:= ncST_END; //Trigger
	CamSeqPara.Configuration.State[2].Event[0].Attribute 			:= ncST_END; //Reaction
	CamSeqPara.Configuration.State[2].Event[0].NextState 			:= 3; //Next State

	(*************************** STATE 3 ****************************)
	CamSeqPara.Configuration.State[3].CamProfileIndex 				:= 16#FFFE;
	CamSeqPara.Configuration.State[3].MasterFactor 					:= 1; //Master Dist.
	CamSeqPara.Configuration.State[3].SlaveFactor 					:= 1; //Slave Dist.

	CamSeqPara.Configuration.State[3].CompMode   	 				:= ncONLYCOMP;
	CamSeqPara.Configuration.State[3].MasterCompDistance			:= 1620; //Master Dist.
	CamSeqPara.Configuration.State[3].SlaveCompDistance				:= 1620; //Slave Dist.

	(** Event **)
	CamSeqPara.Configuration.State[3].Event[0].Type 				:= ncST_END; //Trigger
	CamSeqPara.Configuration.State[3].Event[0].Attribute 			:= ncST_END; //Reaction
	CamSeqPara.Configuration.State[3].Event[0].NextState 			:= 1; //Next State
END_ACTION
```

#### Exercise5.st
```iecst
ACTION Exercise5:

	CamSeqPara.Configuration.Master 			:= ADR(gAxis04);
	CamSeqPara.Configuration.MasterParID 		:= ACP10PAR_PCTRL_S_ACT;

	(** Event 0 - WAIT FOR TRIGGER **)
	CamSeqPara.Configuration.State[0].Event[0].Type 				:= ncST_END; //Trigger
	CamSeqPara.Configuration.State[0].Event[0].Attribute		 	:= ncST_END; //Reaction
	CamSeqPara.Configuration.State[0].Event[0].NextState 			:= 1; //Next State
	(*************************** STATE 1 ****************************)
	CamSeqPara.Configuration.State[1].CamProfileIndex 		  		:= 16#FFFE;
	CamSeqPara.Configuration.State[1].MasterFactor 					:= 1; //Master Dist.
	CamSeqPara.Configuration.State[1].SlaveFactor 					:= 1; //Slave Dist.

	CamSeqPara.Configuration.State[1].CompMode   	 				:= ncONLYCOMP;
	CamSeqPara.Configuration.State[1].MasterCompDistance			:= 1580; //Master Dist.
	CamSeqPara.Configuration.State[1].SlaveCompDistance				:= 1580; //Slave Dist.

	(** Event **)
	CamSeqPara.Configuration.State[1].Event[0].Type 				:= ncST_END; //Trigger
	CamSeqPara.Configuration.State[1].Event[0].Attribute 			:= ncST_END; //Reaction
	CamSeqPara.Configuration.State[1].Event[0].NextState 			:= 2; //Next State

	(*************************** STATE 2 ****************************)
	CamSeqPara.Configuration.State[2].CamProfileIndex 				:= 16#FFFF;
	CamSeqPara.Configuration.State[2].MasterFactor 					:= 400;  //Master Dist.
	CamSeqPara.Configuration.State[2].SlaveFactor 					:= -400; //Slave Dist.

	(** Event **)
	CamSeqPara.Configuration.State[2].Event[0].Type 				:= ncST_END; //Trigger
	CamSeqPara.Configuration.State[2].Event[0].Attribute 			:= ncST_END; //Reaction
	CamSeqPara.Configuration.State[2].Event[0].NextState 			:= 0; //Next State

	(*************************** STATE 3 ****************************)
	CamSeqPara.Configuration.State[3].CamProfileIndex 				:= 16#FFFE;
	CamSeqPara.Configuration.State[3].MasterFactor 					:= 1; //Master Dist.
	CamSeqPara.Configuration.State[3].SlaveFactor 					:= 1; //Slave Dist.

	CamSeqPara.Configuration.State[3].CompMode   	 				:= ncONLYCOMP;
	CamSeqPara.Configuration.State[3].MasterCompDistance			:= 1620; //Master Dist.
	CamSeqPara.Configuration.State[3].SlaveCompDistance				:= 1620; //Slave Dist.

	(** Event **)
	CamSeqPara.Configuration.State[3].Event[0].Type 				:= ncST_END; //Trigger
	CamSeqPara.Configuration.State[3].Event[0].Attribute 			:= ncST_END; //Reaction
	CamSeqPara.Configuration.State[3].Event[0].NextState 			:= 4; //Next State

	(*************************** STATE 4 ****************************)
	CamSeqPara.Configuration.State[4].CamProfileIndex 				:= 16#FFFF;
	CamSeqPara.Configuration.State[4].MasterFactor 					:= 360;  //Master Dist.
	CamSeqPara.Configuration.State[4].SlaveFactor 					:= -360; //Slave Dist.

	(** Event **)
	CamSeqPara.Configuration.State[4].Event[0].Type 				:= ncST_END; //Trigger
	CamSeqPara.Configuration.State[4].Event[0].Attribute 			:= ncST_END; //Reaction
	CamSeqPara.Configuration.State[4].Event[0].NextState 			:= 1; //Next State
END_ACTION
```

Listed in the project but not available here: Logical/Global.typ
